INTERFACE I_AnalogOutput

END_INTERFACE

(* stored: Version 1.1.0.1, ProductVersion 3.1.4026.18
   Itf I_AnalogOutput: Id {fb9ebf89-baf9-4f5d-9f59-8ab21d4a4475} *)
